TYPE "PPrf_A0301_Trasporto"
VERSION : 0.1
// Block: PPrf_A0301_Trasporto
   STRUCT
      VelOvr_PLen_UpTo_1000 : Real;
      VelOvr_PLen_UpTo_1500 : Real;
      VelOvr_PLen_UpTo_2000 : Real;
      VelOvr_PLen_UpTo_2500 : Real;
      VelOvr_PLen_UpTo_3000 : Real;
      VelOvr_PLen_UpTo_3500 : Real;
      VelOvr_PLen_UpTo_4000 : Real;
      VelOvr_PLen_UpTo_4500 : Real;
      VelOvr_PLen_UpTo_5000 : Real;
      VelOvr_PLen_UpTo_5500 : Real;
   END_STRUCT;

END_TYPE
